PROGRAM ldrMain


// Notes
//  I imagine that the control loops can run as independent threads/tasks under the main PlcTask
//  xmeas, xmv, r, and maybe others could be stored in a GVL 
VAR
	
	// data acquitistion from IO blocks
	xmeas_acquire: fb_xmeas_acquire;

	// Molar Percent G control loop
	//pct_g_dpi: fb_discrete_pi		  := (kc:=1, ti:=0.001/60, Ts:=g_Ts_base, hi :=100, lo:=0, x0:=Eadj_0);
	
	// production rate control loop
	prod_rate_loop: fb_prod_rate_ctrl := (kc:=3.2, ti:=120/60, ts:=g_Ts_base, x0:=0, hi:=30, lo:=0);	
	
	// feed ratio control loop
	feed_ratio_ctrl: fb_feed_ratio_ctrl;
	
	// process levels/invetory controller
	level_ctrl: fb_level_ctrl;
		
	// product comnposition controller
	prod_comp_ctrl: fb_prod_comp_ctrl;
	
	// A & C ratio controller
	ac_ratio_ctrl: fb_ac_ratio_ctrl;
	
	// temperature controller
	temp_ctrl: fb_temp_ctrl;
	
	// simulated measurements for debug
	xmeas_simulated: fb_xmeas_simulated;
END_VAR

VAR_INPUT
	
END_VAR
VAR // added by the converter: edge detectors and wires of the graphical bodies
    _w1 : BOOL;
END_VAR

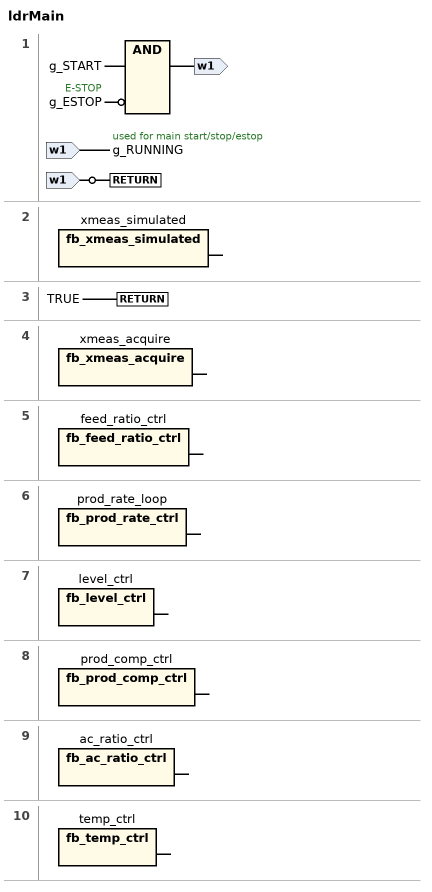
// NETWORK 1
//   g_ESTOP: E-STOP
//   g_RUNNING: used for main start/stop/estop
_w1 := g_START AND NOT g_ESTOP;
g_RUNNING := _w1;
IF NOT _w1 THEN RETURN; END_IF

// NETWORK 2
//   xmeas_simulated: simulated measurements for debug
xmeas_simulated(); // fb_xmeas_simulated

// NETWORK 3
RETURN;

// NETWORK 4
//   xmeas_acquire: data acquitistion from IO blocks
xmeas_acquire(); // fb_xmeas_acquire

// NETWORK 5
//   feed_ratio_ctrl: feed ratio control loop
feed_ratio_ctrl(); // fb_feed_ratio_ctrl

// NETWORK 6
//   prod_rate_loop: Molar Percent G control loop pct_g_dpi: fb_discrete_pi := (kc:=1, ti:=0.001/60, Ts:=g_Ts_base, hi :=100, lo:=0, x0:=Eadj_0); production rate control loop
prod_rate_loop(); // fb_prod_rate_ctrl

// NETWORK 7
//   level_ctrl: process levels/invetory controller
level_ctrl(); // fb_level_ctrl

// NETWORK 8
//   prod_comp_ctrl: product comnposition controller
prod_comp_ctrl(); // fb_prod_comp_ctrl

// NETWORK 9
//   ac_ratio_ctrl: A & C ratio controller
ac_ratio_ctrl(); // fb_ac_ratio_ctrl

// NETWORK 10
//   temp_ctrl: temperature controller
temp_ctrl(); // fb_temp_ctrl

END_PROGRAM

(* stored: Version 1.1.0.1, ProductVersion 3.1.0.26
   POU ldrMain: Id {2b4bc59a-59cf-4d59-b1b8-494101288844} *)
